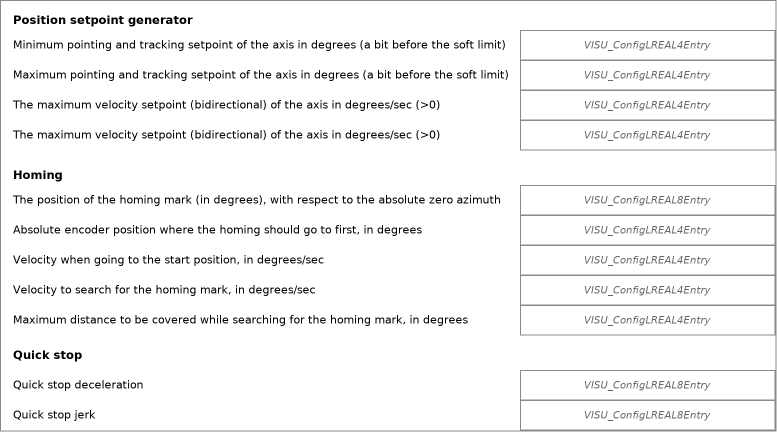
VISUALIZATION VISU_AxesConfig_Elevation_2  // 777x432
VAR_IN_OUT
    active : AxesElevationConfig;
    editable : AxesElevationConfig;
END_VAR
    Frame (520,185 255x30)
        shows VISU_ConfigLREAL8Entry(active := active.homingHomePosition, editable := editable.homingHomePosition)
    Label (10,185 500x30), "The position of the homing mark (in degrees), with respect to the absolute zero azimuth"
    Label (10,5 205x30), "Position setpoint generator"
    Label (10,30 490x30), "Minimum pointing and tracking setpoint of the axis in degrees (a bit before the soft limit)"
    Label (10,60 500x30), "Maximum pointing and tracking setpoint of the axis in degrees (a bit before the soft limit)"
    Label (10,90 475x30), "The maximum velocity setpoint (bidirectional) of the axis in degrees/sec (>0)"
    Label (10,120 475x30), "The maximum velocity setpoint (bidirectional) of the axis in degrees/sec (>0)"
    Label (10,160 205x30), "Homing"
    Label (10,215 475x30), "Absolute encoder position where the homing should go to first, in degrees"
    Label (10,245 475x30), "Velocity when going to the start position, in degrees/sec"
    Label (10,275 505x30), "Velocity to search for the homing mark, in degrees/sec"
    Label (10,305 500x30), "Maximum distance to be covered while searching for the homing mark, in degrees"
    Frame (520,30 255x30)
        shows VISU_ConfigLREAL4Entry(active := active.minPositionSetpoint, editable := editable.minPositionSetpoint)
    Frame (520,60 255x30)
        shows VISU_ConfigLREAL4Entry(active := active.maxPositionSetpoint, editable := editable.maxPositionSetpoint)
    Frame (520,90 255x30)
        shows VISU_ConfigLREAL4Entry(active := active.maxVelocitySetpoint, editable := editable.maxVelocitySetpoint)
    Frame (520,120 255x30)
        shows VISU_ConfigLREAL4Entry(active := active.maxAccelerationSetpoint, editable := editable.maxAccelerationSetpoint)
    Frame (520,215 255x30)
        shows VISU_ConfigLREAL4Entry(active := active.homingStartAbsEncPosition, editable := editable.homingStartAbsEncPosition)
    Frame (520,245 255x30)
        shows VISU_ConfigLREAL4Entry(active := active.homingGotoStartVelocity, editable := editable.homingGotoStartVelocity)
    Frame (520,275 255x30)
        shows VISU_ConfigLREAL4Entry(active := active.homingVelocity, editable := editable.homingVelocity)
    Frame (520,305 255x30)
        shows VISU_ConfigLREAL4Entry(active := active.homingRange, editable := editable.homingRange)
    Label (10,340 205x30), "Quick stop"
    Frame (520,370 255x30)
        shows VISU_ConfigLREAL8Entry(active := active.quickStopDeceleration, editable := editable.quickStopDeceleration)
    Label (10,370 500x30), "Quick stop deceleration"
    Label (10,400 500x30), "Quick stop jerk"
    Frame (520,400 255x30)
        shows VISU_ConfigLREAL8Entry(active := active.quickStopJerk, editable := editable.quickStopJerk)
END_VISUALIZATION

(* stored: Version 1.1.0.1, ProductVersion 3.1.4019.2
   Visu VISU_AxesConfig_Elevation_2: Id {e5cd39f3-26b9-4e26-9714-db97592ce1c4} *)
